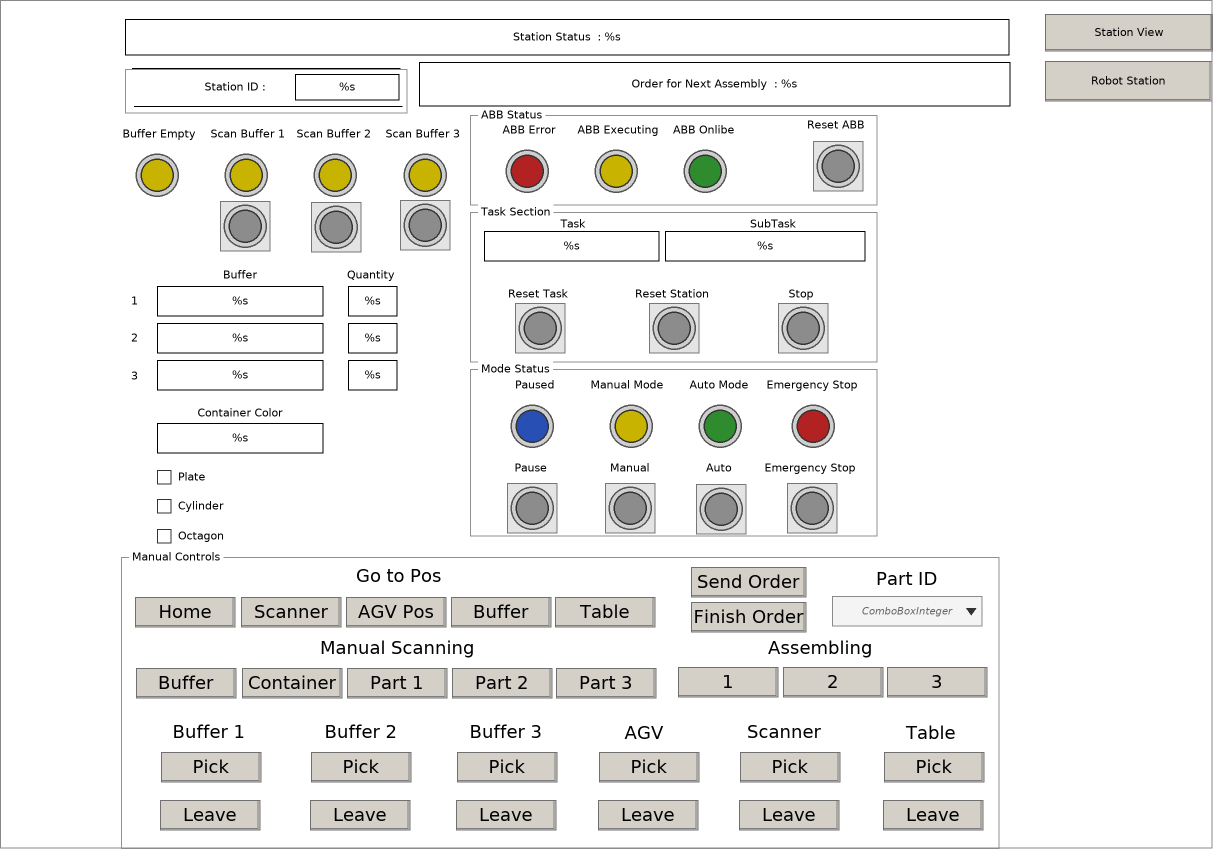
VISUALIZATION Visualization  // 1213x849
    Rectangle (125,19 884x36), "Station Status : %s", text variable: Visualaisation_Control.mxStationStatus
    GroupBox (125,61 282x52)
        Line (7,7) (275,7)
        Label (35,11 150x30), "Station ID :"
        Rectangle (170,13 104x26), "%s", text variable: GVL.mwStationID
        Line (9,45) (277,45)
    Button (1045,61 167x40), "Robot Station"
        OnMouseClick: change screen: RobotStation
    Rectangle (419,62 591x44), "Order for Next Assembly : %s", text variable: GVL.qsOrderFornextAssembly
    Button (1045,14 168x37), "Station View"
        OnMouseClick: change screen: Station
    Lamp1 (132,150 50x50), variable: MAIN.ixEmptyBuffer, style: Lamp-Lamp1-Yellow
    Label (84,119 150x30), "Buffer Empty"
    Lamp1 (221,150 50x50), style: Lamp-Lamp1-Yellow
    Label (173,119 150x30), "Scan Buffer 1"
    Lamp1 (310,150 50x50), style: Lamp-Lamp1-Yellow
    Label (259,119 150x30), "Scan Buffer 2"
    Lamp1 (400,150 50x50), style: Lamp-Lamp1-Yellow
    Label (348,119 150x30), "Scan Buffer 3"
    GroupBox (470,107 407x98), "ABB Status"
        PushSwitch (343,34 50x50), variable: MAIN.ixResetABB, behaviour: TAP, style: Switch-PushSwitch-Gray
        Label (291,3 150x30), "Reset ABB"
    Lamp1 (502,146 50x50), variable: MAIN.qxABBErrorLamp, style: Lamp-Lamp1-Red
    Label (454,115 150x30), "ABB Error"
    Lamp1 (591,146 50x50), variable: MAIN.qxABBExecutLamp, style: Lamp-Lamp1-Yellow
    Label (543,115 150x30), "ABB Executing"
    Lamp1 (680,146 50x50), variable: MAIN.qxABBonlineLamp, style: Lamp-Lamp1-Green
    Label (629,115 150x30), "ABB Onlibe"
    GroupBox (470,204 407x158), "Task Section"
        Rectangle (14,27 175x30), "%s", text variable: MAIN.qsTask
        Rectangle (195,27 200x30), "%s", text variable: MAIN.qsSubTask
        PushSwitch (179,99 50x50), behaviour: TAP, style: Switch-PushSwitch-Gray
        PushSwitch (308,99 50x50), behaviour: TAP, style: Switch-PushSwitch-Gray
    Label (498,209 150x30), "Task"
    Label (698,209 150x30), "SubTask"
    PushSwitch (515,303 50x50), behaviour: TAP, style: Switch-PushSwitch-Gray
    Label (463,279 150x30), "Reset Task"
    Label (597,279 150x30), "Reset Station"
    Label (726,279 150x30), "Stop"
    GroupBox (470,361 407x175), "Mode Status"
        PushSwitch (37,122 50x50), variable: MAIN.ixPauseButt, behaviour: TOGGLE, style: Switch-PushSwitch-Gray
        PushSwitch (135,122 50x50), variable: MAIN.qxManualMode, behaviour: TAP, style: Switch-PushSwitch-Gray
        PushSwitch (226,123 50x50), variable: MAIN.qxAutoMode, behaviour: TAP, style: Switch-PushSwitch-Gray
        PushSwitch (317,122 50x50), variable: GVL.ixEmergencyStop, behaviour: TOGGLE, style: Switch-PushSwitch-Gray
        Label (174,92 150x30), "Auto"
        Label (265,92 150x30), "Emergency Stop"
    Lamp1 (507,401 50x50), variable: MAIN.qxPauseLamp, style: Lamp-Lamp1-Blue
    Label (460,370 150x30), "Paused"
    Lamp1 (606,401 50x50), variable: MAIN.ixManualLamp, style: Lamp-Lamp1-Yellow
    Label (552,370 150x30), "Manual Mode"
    Lamp1 (695,401 50x50), variable: MAIN.ixAutoLamp, style: Lamp-Lamp1-Green
    Label (644,370 150x30), "Auto Mode"
    Lamp1 (788,401 50x50), variable: MAIN.qxEmergySTLamp, style: Lamp-Lamp1-Red
    Label (737,370 150x30), "Emergency Stop"
    Label (456,453 150x30), "Pause"
    Label (555,453 150x30), "Manual"
    Rectangle (157,286 166x30), "%s", text variable: GVL.BufferProducts.Storage1.Component
    Rectangle (348,286 49x30), "%s", text variable: GVL.BufferProducts.Storage1.Quatity
    Rectangle (157,323 166x30), "%s", text variable: GVL.BufferProducts.Storage2.Component
    Rectangle (348,323 49x30), "%s", text variable: GVL.BufferProducts.Storage2.Quatity
    Rectangle (157,360 166x30), "%s", text variable: GVL.BufferProducts.Storage3.Component
    Rectangle (348,360 49x30), "%s", text variable: GVL.BufferProducts.Storage3.Quatity
    PushSwitch (220,201 50x50), behaviour: TAP, style: Switch-PushSwitch-Gray
    PushSwitch (311,202 50x50), behaviour: TAP, style: Switch-PushSwitch-Gray
    PushSwitch (400,200 50x50), behaviour: TAP, style: Switch-PushSwitch-Gray
    Label (165,260 150x30), "Buffer"
    Label (296,260 150x30), "Quantity"
    Label (116,286 37x30), "1"
    Label (116,323 37x30), "2"
    Label (116,361 37x30), "3"
    Rectangle (157,423 166x30), "%s", text variable: MAIN.qsContainer
    Label (165,398 150x30), "Container Color"
    Checkbox (155,462 150x30), "Plate", variable: MAIN.mxPlateAvailable
    Checkbox (155,491 150x30), "Cylinder", variable: MAIN.mxCylinderAvailable
    Checkbox (155,521 150x30), "Octagon", variable: MAIN.mxOctagonAvailable
    GroupBox (121,549 878x300), "Manual Controls"
        Button (14,48 100x30), "Home"
            tap ABB_Control_FB.ixGotoHome
        Button (120,48 100x30), "Scanner"
            tap ABB_Control_FB.ixGotoScanner
        Button (225,48 100x30), "AGV Pos"
            tap ABB_Control_FB.ixGotoAGV
        Button (330,48 100x30), "Buffer"
            tap ABB_Control_FB.ixGotoBuffer
        Button (434,48 100x30), "Table"
            tap ABB_Control_FB.ixGotoTable
        Button (15,119 100x30), "Buffer"
            tap ABB_Control_FB.ixScanBuffer
        Label (95,12 366x30), "Go to Pos"
        Label (95,84 363x30), "Manual Scanning"
        ComboBoxInteger (711,47 150x30), variable: MAIN.mwPartID, text list: MAIN.sPartID
        Label (695,16 182x28), "Part ID"
        Label (518,84 363x30), "Assembling"
        Button (557,118 100x30), "1"
            toggle ABB_Control_FB.ixAssemble1
        Button (40,203 100x30), "Pick"
            tap ABB_Control_FB.ixPickBuffer1
        Button (478,203 100x30), "Pick"
            tap ABB_Control_FB.ixPickAGV
        Button (619,203 100x30), "Pick"
            tap ABB_Control_FB.ixPickScanner
        Button (336,203 100x30), "Pick"
            tap ABB_Control_FB.ixPickBuffer3
        Button (190,203 100x30), "Pick"
            tap ABB_Control_FB.ixPickBuffer2
        Button (39,251 100x30), "Leave"
            tap ABB_Control_FB.ixLeaveBuffer1
        Label (13,168 150x30), "Buffer 1"
        Label (165,168 150x30), "Buffer 2"
        Label (310,168 150x30), "Buffer 3"
        Label (448,169 150x30), "AGV"
        Label (588,168 150x30), "Scanner"
        Label (735,169 150x30), "Table"
        Button (570,18 115x30), "Send Order"
            tap ABB_Control_FB.ixSendOrder
        Button (570,53 115x30), "Finish Order"
            tap ABB_Control_FB.ixFinishOrder
    Label (1062,118 150x30)
    Button (242,668 100x30), "Container"
        tap ABB_Control_FB.ixScanContainer
    Button (347,668 100x30), "Part 1"
        toggle ABB_Control_FB.ixScanPart1
    Button (452,668 100x30), "Part 2"
        toggle ABB_Control_FB.ixScanPart2
    Button (556,668 100x30), "Part 3"
        toggle ABB_Control_FB.ixScanPart3
    Button (783,667 100x30), "2"
        toggle ABB_Control_FB.ixAssemble2
    Button (887,667 100x30), "3"
        toggle ABB_Control_FB.ixAssemble3
    Button (884,752 100x30), "Pick"
        tap ABB_Control_FB.ixPickTable
    Button (598,800 100x30), "Leave"
        tap ABB_Control_FB.ixLeaveAGV
    Button (739,800 100x30), "Leave"
        tap ABB_Control_FB.ixLeaveScanner
    Button (456,800 100x30), "Leave"
        tap ABB_Control_FB.ixLeaveBuffer3
    Button (310,800 100x30), "Leave"
        tap ABB_Control_FB.ixLeaveBuffer2
    Button (883,800 100x30), "Leave"
        tap ABB_Control_FB.ixLeaveTable
END_VISUALIZATION

(* stored: Version 1.1.0.1, ProductVersion 3.1.4024.12
   Visu Visualization: Id {08c1f753-3e44-4c26-b458-35ef78727ab8} *)
